// TIA Portal project "TIA_PORTAL_SORTING_STATION" (V20)

(* hardware
DEVICE "S7-1200 station_1"  S7-1200 Station
   slot 0: "Rack_0"  S7-1200 Rack  Rack  V1.0
   slot 1: "PLC_1"  CPU 1214C AC/DC/Rly  6ES7 214-1BG40-0XB0  V4.1
*)

// ===== PLC "PLC_1"  CPU 1214C AC/DC/Rly =====

VAR_GLOBAL   // PLC tag table "Default tag table"
   "Sensor_Pieza" AT %I0.0 : Bool;
   "CINTA" AT %Q0.0 : Bool;
   "S_LASER_RAMPA" AT %I0.2 : Bool;
   "Llave" AT %I0.7 : Bool;
   "START" AT %I1.2 : Bool;
   "M_STARTING" AT %M2.1 : Bool;
   "SENSOR_SERVO1" AT %I0.1 : Bool;
   "SENSOR_SERVO2" AT %I0.3 : Bool;
   "System_Byte" AT %MB300 : Byte;
   "FirstScan" AT %M300.0 : Bool;
   "DiagStatusUpdate" AT %M300.1 : Bool;
   "AlwaysTRUE" AT %M300.2 : Bool;
   "AlwaysFALSE" AT %M300.3 : Bool;
   "SIEMPRE_CERO" AT %M0.0 : Bool;
   "SIEMPRE_UNO" AT %M0.1 : Bool;
   "M_STOPPED" AT %M2.0 : Bool;
   "M_STARTED" AT %M2.2 : Bool;
   "M_STOPPING" AT %M2.3 : Bool;
   "M_ABORTING" AT %M2.4 : Bool;
   "M_RESET" AT %M2.5 : Bool;
   "M_FIN_CICLO" AT %M2.6 : Bool;
   "RESET" AT %I1.1 : Bool;
   "STOP" AT %I1.0 : Bool;
   "IR_A_M_STOPPED" AT %M4.3 : Bool;
   "PILOTO_START" AT %Q0.4 : Bool;
   "PILOTO_RESET" AT %Q0.5 : Bool;
   "Q1_STOPPED" AT %Q0.6 : Bool;
   "Q2_EMEG" AT %Q0.7 : Bool;
   "Timer_1" AT %M5.0 : Bool;
   "Tag_3" AT %M6.0 : Bool;
   "Intermitente" AT %M6.1 : Bool;
   "M_CINTA" AT %M3.0 : Bool;
   "Tag_1" AT %MB3 : Byte;
   "M_INICIO_RESET" AT %M4.2 : Bool;
   "M_FIN_RESET" AT %M4.1 : Bool;
   "M_SERVO_1" AT %M3.1 : Bool;
   "M_SERVO_2" AT %M3.2 : Bool;
   "M_PISTON" AT %M3.3 : Bool;
   "START_TIMER" AT %M5.1 : Bool;
   "M_INICIO_SECUENCIA" AT %M3.4 : Bool;
   "S_BARRERA" AT %I0.6 : Bool;
   "S_CANCELA_NEGRO" AT %I0.5 : Bool;
   "S_PIEZA_METALICA" AT %I0.4 : Bool;
   "SERVO_1" AT %Q0.1 : Bool;
   "SERVO_2" AT %Q0.2 : Bool;
   "PISTON" AT %Q0.3 : Bool;
   "M_PIEZA" AT %M3.5 : Bool;
   "Tag_2" AT %MW100 : Int;
   "M_TOTAL_ROJO" AT %M2.7 : Bool;
   "M_TOTAL_METAL" AT %M4.0 : Bool;
   "Tag_4" AT %MW101 : Int;
   "M_ROJO" AT %M7.0 : Bool;
   "M_BANDA_R" AT %M7.1 : Bool;
   "Tag_5" AT %MW102 : Int;
   "Tag_6" AT %MW107 : Int;
   "Tag_7" AT %MB7 : Byte;
   "Tag_8" AT %MB4 : Byte;
   "Tag_9" AT %MB5 : Byte;
   "M_Negro" AT %M7.2 : Bool;
END_VAR

VAR_GLOBAL   // PLC tag table "Tag table_1"
   "Clock_Byte" AT %MB100 : Byte;
   "Clock_10Hz" AT %M100.0 : Bool;
   "Clock_5Hz" AT %M100.1 : Bool;
   "Clock_2.5Hz" AT %M100.2 : Bool;
   "Clock_2Hz" AT %M100.3 : Bool;
   "Clock_1.25Hz" AT %M100.4 : Bool;
   "Clock_1Hz" AT %M100.5 : Bool;
   "Clock_0.625Hz" AT %M100.6 : Bool;
   "Clock_0.5Hz" AT %M100.7 : Bool;
END_VAR

// folder: System blocks/Program resources

DATA_BLOCK "IEC_Timer_0_DB"   // DB1
{ S7_Optimized_Access := 'TRUE' }
AUTHOR : Simatic
FAMILY : IEC
NAME : IEC_TMR
VERSION : 1.0
// stored: InstanceOfName IEC_TIMER
"IEC_TIMER"
BEGIN
END_DATA_BLOCK

DATA_BLOCK "IEC_Timer_0_DB_1"   // DB2
{ S7_Optimized_Access := 'TRUE' }
AUTHOR : Simatic
FAMILY : IEC
NAME : IEC_TMR
VERSION : 1.0
// stored: InstanceOfName IEC_TIMER
"IEC_TIMER"
BEGIN
END_DATA_BLOCK

DATA_BLOCK "IEC_Timer_0_DB_2"   // DB3
{ S7_Optimized_Access := 'TRUE' }
AUTHOR : Simatic
FAMILY : IEC
NAME : IEC_TMR
VERSION : 1.0
// stored: InstanceOfName IEC_TIMER
"IEC_TIMER"
BEGIN
END_DATA_BLOCK

DATA_BLOCK "IEC_Timer_0_DB_3"   // DB4
{ S7_Optimized_Access := 'TRUE' }
AUTHOR : Simatic
FAMILY : IEC
NAME : IEC_TMR
VERSION : 1.0
// stored: InstanceOfName IEC_TIMER
"IEC_TIMER"
BEGIN
END_DATA_BLOCK

DATA_BLOCK "IEC_Timer_0_DB_4"   // DB5
{ S7_Optimized_Access := 'TRUE' }
AUTHOR : Simatic
FAMILY : IEC
NAME : IEC_TMR
VERSION : 1.0
// stored: InstanceOfName IEC_TIMER
"IEC_TIMER"
BEGIN
END_DATA_BLOCK

DATA_BLOCK "IEC_Timer_0_DB_5"   // DB6
{ S7_Optimized_Access := 'TRUE' }
AUTHOR : Simatic
FAMILY : IEC
NAME : IEC_TMR
VERSION : 1.0
// stored: InstanceOfName IEC_TIMER
"IEC_TIMER"
BEGIN
END_DATA_BLOCK

DATA_BLOCK "IEC_Timer_0_DB_6"   // DB7
{ S7_Optimized_Access := 'TRUE' }
AUTHOR : Simatic
FAMILY : IEC
NAME : IEC_TMR
VERSION : 1.0
// stored: InstanceOfName IEC_TIMER
"IEC_TIMER"
BEGIN
END_DATA_BLOCK

DATA_BLOCK "IEC_Timer_0_DB_7"   // DB8
{ S7_Optimized_Access := 'TRUE' }
AUTHOR : Simatic
FAMILY : IEC
NAME : IEC_TMR
VERSION : 1.0
// stored: InstanceOfName IEC_TIMER
"IEC_TIMER"
BEGIN
END_DATA_BLOCK

DATA_BLOCK "IEC_Counter_0_DB"   // DB10
{ S7_Optimized_Access := 'TRUE' }
AUTHOR : Simatic
FAMILY : IEC
NAME : CNTR
VERSION : 1.0
// stored: InstanceOfName IEC_COUNTER
"IEC_COUNTER"
BEGIN
END_DATA_BLOCK

DATA_BLOCK "IEC_Counter_0_DB_1"   // DB11
{ S7_Optimized_Access := 'TRUE' }
AUTHOR : Simatic
FAMILY : IEC
NAME : CNTR
VERSION : 1.0
// stored: InstanceOfName IEC_COUNTER
"IEC_COUNTER"
BEGIN
END_DATA_BLOCK

DATA_BLOCK "IEC_Counter_0_DB_2"   // DB12
{ S7_Optimized_Access := 'TRUE' }
AUTHOR : Simatic
FAMILY : IEC
NAME : CNTR
VERSION : 1.0
// stored: InstanceOfName IEC_COUNTER
"IEC_COUNTER"
BEGIN
END_DATA_BLOCK

// folder: (top level)

FUNCTION "RESET_ESTADO" : Void   // FC1, LAD
{ S7_Optimized_Access := 'TRUE' }
VERSION : 0.1
BEGIN

REGION Network 1
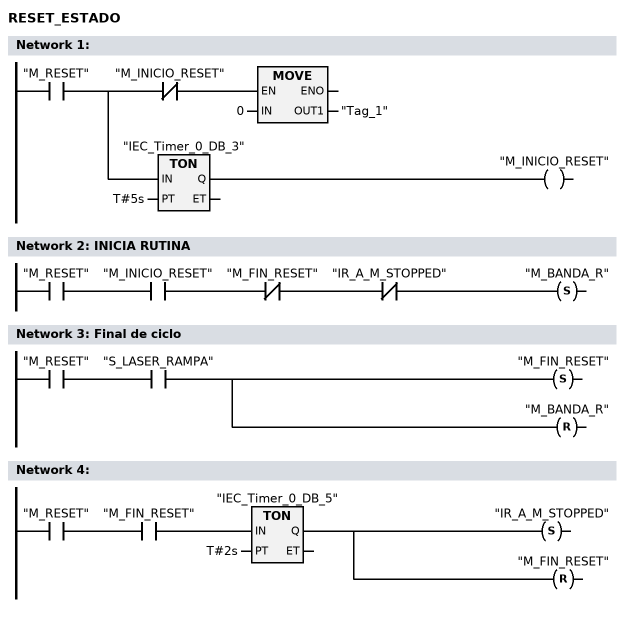
   IF "M_RESET" AND NOT "M_INICIO_RESET" THEN "Tag_1" := 0; END_IF;
   "IEC_Timer_0_DB_3".TON(IN := "M_RESET", PT := T#5s);
   "M_INICIO_RESET" := "IEC_Timer_0_DB_3".Q;
END_REGION

REGION Network 2: INICIA RUTINA
   RUNG wire#powerrail
      Contact( "M_RESET" )
      Contact( "M_INICIO_RESET" )
      I_Contact( "M_FIN_RESET" )
      I_Contact( "IR_A_M_STOPPED" )
      S_Coil( "M_BANDA_R" )
   END_RUNG
   // the same network as SCL:
   IF "M_RESET" AND "M_INICIO_RESET" AND NOT "M_FIN_RESET" AND NOT "IR_A_M_STOPPED" THEN
       "M_BANDA_R" := TRUE;
   END_IF;
END_REGION

REGION Network 3: Final de ciclo
   RUNG wire#powerrail
      Contact( "M_RESET" )
      Contact( "S_LASER_RAMPA" )
      wire#w1
      S_Coil( "M_FIN_RESET" )
   END_RUNG
   RUNG wire#w1
      R_Coil( "M_BANDA_R" )
   END_RUNG
   // the same network as SCL:
   IF "M_RESET" AND "S_LASER_RAMPA" THEN
       "M_FIN_RESET" := TRUE;
       "M_BANDA_R" := FALSE;
   END_IF;
END_REGION

REGION Network 4
   "IEC_Timer_0_DB_5".TON(IN := "M_RESET" AND "M_FIN_RESET", PT := T#2s);
   IF "IEC_Timer_0_DB_5".Q THEN
       "IR_A_M_STOPPED" := TRUE;
       "M_FIN_RESET" := FALSE;
   END_IF;
END_REGION
END_FUNCTION

FUNCTION "Maquina_Estado" : Void   // FC2, LAD
{ S7_Optimized_Access := 'TRUE' }
VERSION : 0.1
   VAR_TEMP   // added for the SCL form of the ladder/FBD networks
      _w1 : Bool;
   END_VAR
BEGIN

REGION Network 1: SECUENCIA_STARTING
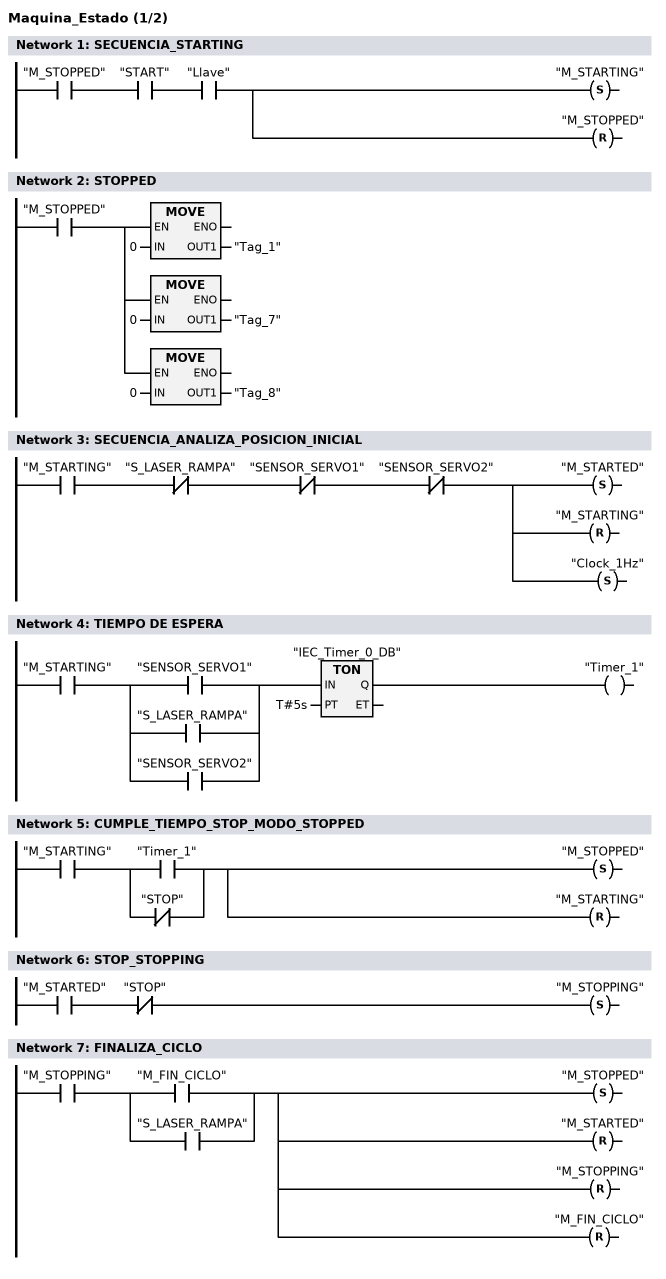
   RUNG wire#powerrail
      Contact( "M_STOPPED" )
      Contact( "START" )
      Contact( "Llave" )
      wire#w1
      S_Coil( "M_STARTING" )
   END_RUNG
   RUNG wire#w1
      R_Coil( "M_STOPPED" )
   END_RUNG
   // the same network as SCL:
   IF "M_STOPPED" AND "START" AND "Llave" THEN
       "M_STARTING" := TRUE;
       "M_STOPPED" := FALSE;
   END_IF;
END_REGION

REGION Network 2: STOPPED
   RUNG wire#powerrail
      Contact( "M_STOPPED" )
      wire#w1
      Move(in := 0, out1 => "Tag_1")
   END_RUNG
   RUNG wire#w1
      Move(in := 0, out1 => "Tag_7")
   END_RUNG
   RUNG wire#w1
      Move(in := 0, out1 => "Tag_8")
   END_RUNG
   // the same network as SCL:
   IF "M_STOPPED" THEN
       "Tag_1" := 0;
       "Tag_7" := 0;
       "Tag_8" := 0;
   END_IF;
END_REGION

REGION Network 3: SECUENCIA_ANALIZA_POSICION_INICIAL
   RUNG wire#powerrail
      Contact( "M_STARTING" )
      I_Contact( "S_LASER_RAMPA" )
      I_Contact( "SENSOR_SERVO1" )
      I_Contact( "SENSOR_SERVO2" )
      wire#w1
      S_Coil( "M_STARTED" )
   END_RUNG
   RUNG wire#w1
      R_Coil( "M_STARTING" )
   END_RUNG
   RUNG wire#w1
      S_Coil( "Clock_1Hz" )
   END_RUNG
   // the same network as SCL:
   IF "M_STARTING" AND NOT "S_LASER_RAMPA" AND NOT "SENSOR_SERVO1" AND NOT "SENSOR_SERVO2" THEN
       "M_STARTED" := TRUE;
   END_IF;
   #_w1 := "M_STARTING" AND NOT "S_LASER_RAMPA" AND NOT "SENSOR_SERVO1" AND NOT "SENSOR_SERVO2";
   IF #_w1 THEN
       "M_STARTING" := FALSE;
       "Clock_1Hz" := TRUE;
   END_IF;
END_REGION

REGION Network 4: TIEMPO DE ESPERA
   "IEC_Timer_0_DB".TON(IN := "M_STARTING" AND ("SENSOR_SERVO1" OR "S_LASER_RAMPA" OR "SENSOR_SERVO2"),
                        PT := T#5s);
   "Timer_1" := "IEC_Timer_0_DB".Q;
END_REGION

REGION Network 5: CUMPLE_TIEMPO_STOP_MODO_STOPPED
   RUNG wire#powerrail
      Contact( "M_STARTING" )
      wire#w1
      Contact( "Timer_1" )
      wire#w2
      S_Coil( "M_STOPPED" )
   END_RUNG
   RUNG wire#w1
      I_Contact( "STOP" )
   END_RUNG wire#w2
   RUNG wire#w2
      R_Coil( "M_STARTING" )
   END_RUNG
   // the same network as SCL:
   IF "M_STARTING" AND ("Timer_1" OR NOT "STOP") THEN
       "M_STOPPED" := TRUE;
       "M_STARTING" := FALSE;
   END_IF;
END_REGION

REGION Network 6: STOP_STOPPING
   RUNG wire#powerrail
      Contact( "M_STARTED" )
      I_Contact( "STOP" )
      S_Coil( "M_STOPPING" )
   END_RUNG
   // the same network as SCL:
   IF "M_STARTED" AND NOT "STOP" THEN "M_STOPPING" := TRUE; END_IF;
END_REGION

REGION Network 7: FINALIZA_CICLO
   RUNG wire#powerrail
      Contact( "M_STOPPING" )
      wire#w1
      Contact( "M_FIN_CICLO" )
      wire#w2
      S_Coil( "M_STOPPED" )
   END_RUNG
   RUNG wire#w1
      Contact( "S_LASER_RAMPA" )
   END_RUNG wire#w2
   RUNG wire#w2
      R_Coil( "M_STARTED" )
   END_RUNG
   RUNG wire#w2
      R_Coil( "M_STOPPING" )
   END_RUNG
   RUNG wire#w2
      R_Coil( "M_FIN_CICLO" )
   END_RUNG
   // the same network as SCL:
   IF "M_STOPPING" AND ("M_FIN_CICLO" OR "S_LASER_RAMPA") THEN
       "M_STOPPED" := TRUE;
       "M_STARTED" := FALSE;
   END_IF;
   #_w1 := "M_STOPPING" AND ("M_FIN_CICLO" OR "S_LASER_RAMPA");
   IF #_w1 THEN
       "M_STOPPING" := FALSE;
       "M_FIN_CICLO" := FALSE;
   END_IF;
END_REGION

REGION Network 8: SI PRESIONA EL PARO DE EMERGENCIA PASAMOS A ABORTING
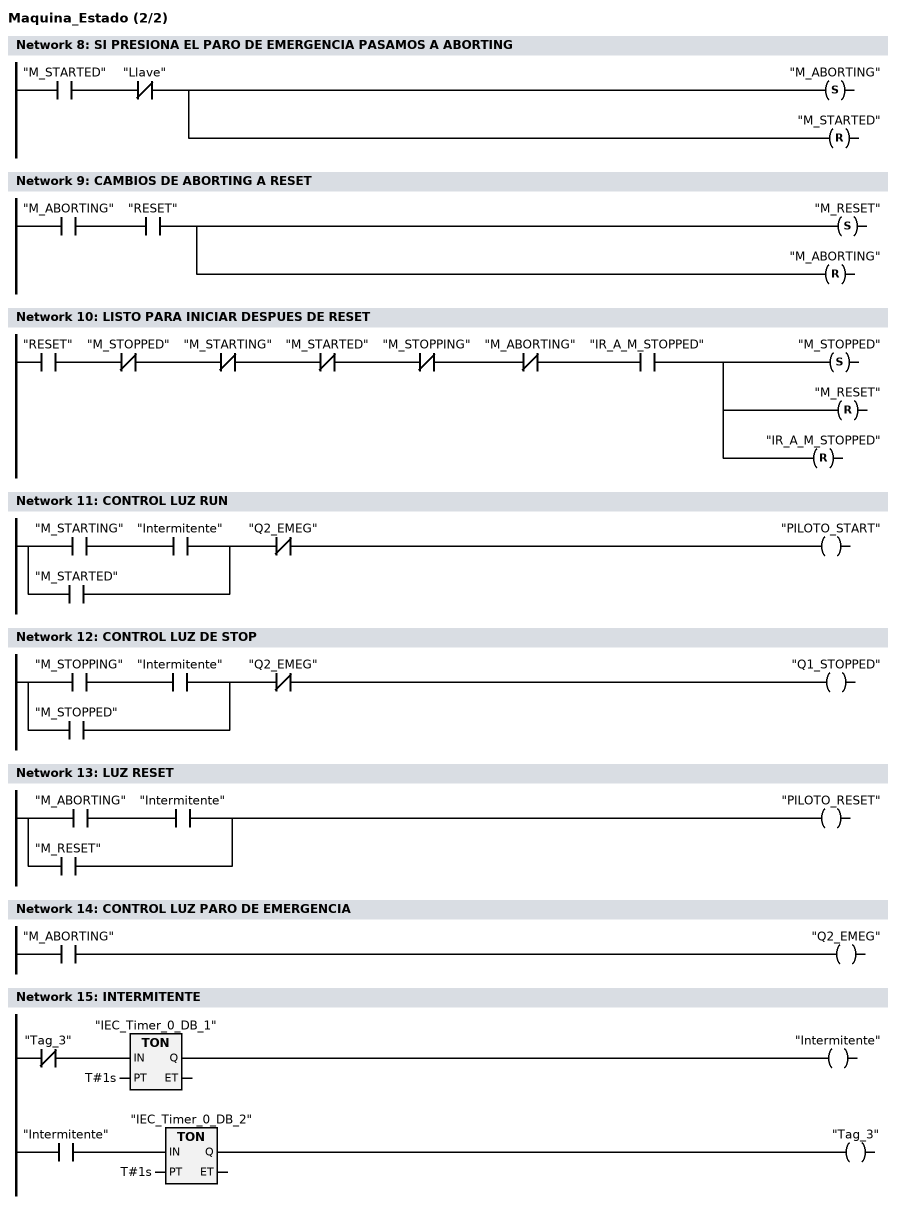
   RUNG wire#powerrail
      Contact( "M_STARTED" )
      I_Contact( "Llave" )
      wire#w1
      S_Coil( "M_ABORTING" )
   END_RUNG
   RUNG wire#w1
      R_Coil( "M_STARTED" )
   END_RUNG
   // the same network as SCL:
   IF "M_STARTED" AND NOT "Llave" THEN
       "M_ABORTING" := TRUE;
       "M_STARTED" := FALSE;
   END_IF;
END_REGION

REGION Network 9: CAMBIOS DE ABORTING A RESET
   RUNG wire#powerrail
      Contact( "M_ABORTING" )
      Contact( "RESET" )
      wire#w1
      S_Coil( "M_RESET" )
   END_RUNG
   RUNG wire#w1
      R_Coil( "M_ABORTING" )
   END_RUNG
   // the same network as SCL:
   IF "M_ABORTING" AND "RESET" THEN
       "M_RESET" := TRUE;
       "M_ABORTING" := FALSE;
   END_IF;
END_REGION

REGION Network 10: LISTO PARA INICIAR DESPUES DE RESET
   RUNG wire#powerrail
      Contact( "RESET" )
      I_Contact( "M_STOPPED" )
      I_Contact( "M_STARTING" )
      I_Contact( "M_STARTED" )
      I_Contact( "M_STOPPING" )
      I_Contact( "M_ABORTING" )
      Contact( "IR_A_M_STOPPED" )
      wire#w1
      S_Coil( "M_STOPPED" )
   END_RUNG
   RUNG wire#w1
      R_Coil( "M_RESET" )
   END_RUNG
   RUNG wire#w1
      R_Coil( "IR_A_M_STOPPED" )
   END_RUNG
   // the same network as SCL:
   #_w1 := "RESET" AND NOT "M_STOPPED" AND NOT "M_STARTING" AND NOT "M_STARTED" AND NOT "M_STOPPING" AND NOT "M_ABORTING" AND "IR_A_M_STOPPED";
   IF #_w1 THEN
       "M_STOPPED" := TRUE;
       "M_RESET" := FALSE;
       "IR_A_M_STOPPED" := FALSE;
   END_IF;
END_REGION

REGION Network 11: CONTROL LUZ RUN
   RUNG wire#powerrail
      Contact( "M_STARTING" )
      Contact( "Intermitente" )
      wire#w1
      I_Contact( "Q2_EMEG" )
      Coil( "PILOTO_START" )
   END_RUNG
   RUNG wire#powerrail
      Contact( "M_STARTED" )
   END_RUNG wire#w1
   // the same network as SCL:
   "PILOTO_START" := (("M_STARTING" AND "Intermitente") OR "M_STARTED") AND NOT "Q2_EMEG";
END_REGION

REGION Network 12: CONTROL LUZ DE STOP
   RUNG wire#powerrail
      Contact( "M_STOPPING" )
      Contact( "Intermitente" )
      wire#w1
      I_Contact( "Q2_EMEG" )
      Coil( "Q1_STOPPED" )
   END_RUNG
   RUNG wire#powerrail
      Contact( "M_STOPPED" )
   END_RUNG wire#w1
   // the same network as SCL:
   "Q1_STOPPED" := (("M_STOPPING" AND "Intermitente") OR "M_STOPPED") AND NOT "Q2_EMEG";
END_REGION

REGION Network 13: LUZ RESET
   RUNG wire#powerrail
      Contact( "M_ABORTING" )
      Contact( "Intermitente" )
      wire#w1
      Coil( "PILOTO_RESET" )
   END_RUNG
   RUNG wire#powerrail
      Contact( "M_RESET" )
   END_RUNG wire#w1
   // the same network as SCL:
   "PILOTO_RESET" := ("M_ABORTING" AND "Intermitente") OR "M_RESET";
END_REGION

REGION Network 14: CONTROL LUZ PARO DE EMERGENCIA
   RUNG wire#powerrail
      Contact( "M_ABORTING" )
      Coil( "Q2_EMEG" )
   END_RUNG
   // the same network as SCL:
   "Q2_EMEG" := "M_ABORTING";
END_REGION

REGION Network 15: INTERMITENTE
   "IEC_Timer_0_DB_1".TON(IN := NOT "Tag_3", PT := T#1s);
   "Intermitente" := "IEC_Timer_0_DB_1".Q;
   "IEC_Timer_0_DB_2".TON(IN := "Intermitente", PT := T#1s);
   "Tag_3" := "IEC_Timer_0_DB_2".Q;
END_REGION
END_FUNCTION

FUNCTION "Programacion secuencia" : Void   // FC3, LAD
{ S7_Optimized_Access := 'TRUE' }
VERSION : 0.1
   VAR_TEMP   // added for the SCL form of the ladder/FBD networks
      _w1 : Bool;
   END_VAR
BEGIN

REGION Network 1: Comprobacion
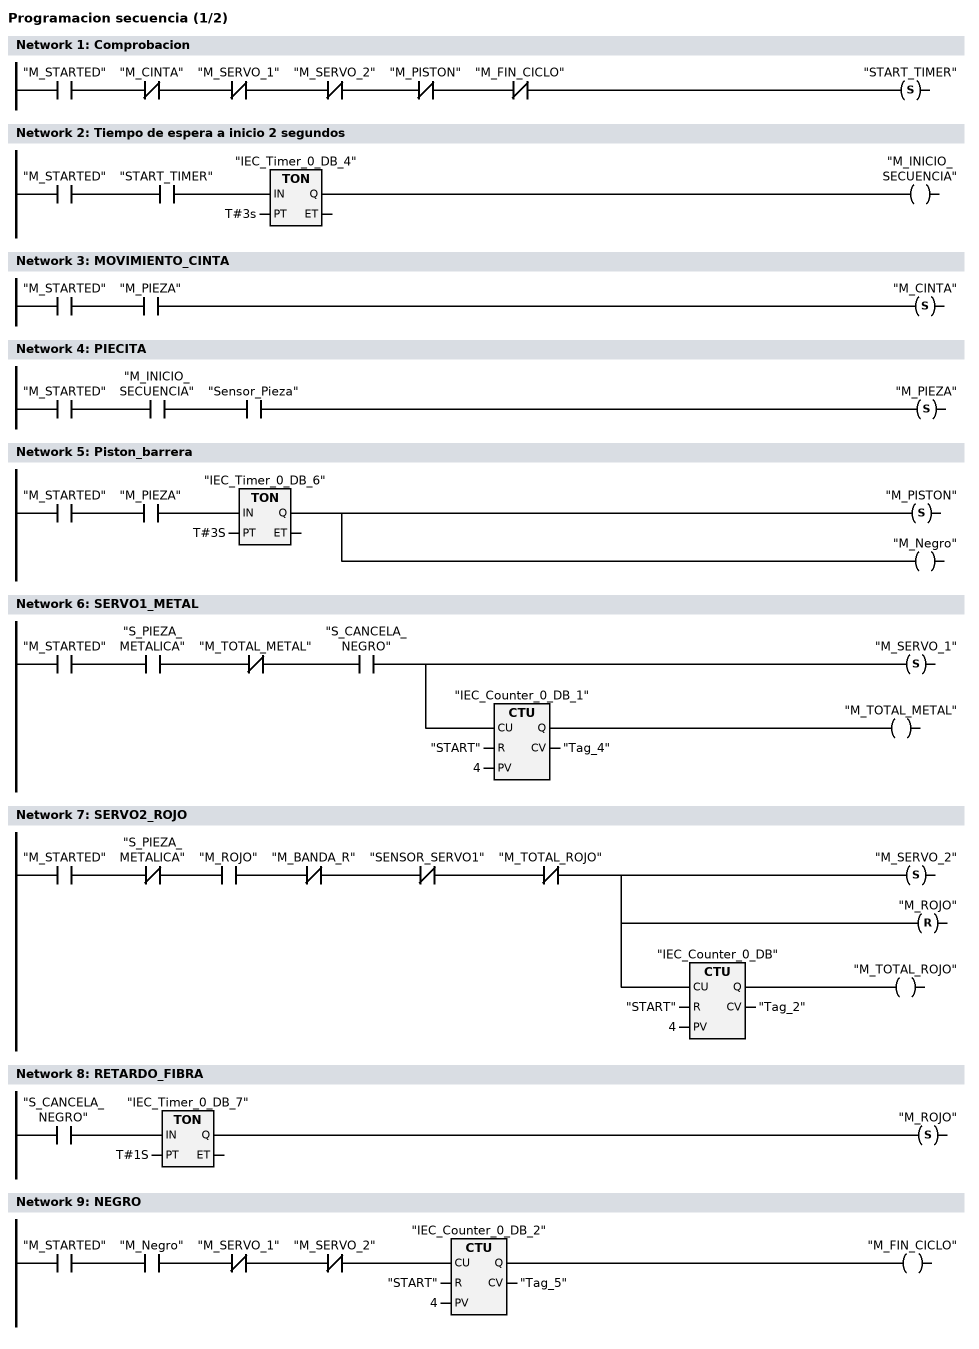
   RUNG wire#powerrail
      Contact( "M_STARTED" )
      I_Contact( "M_CINTA" )
      I_Contact( "M_SERVO_1" )
      I_Contact( "M_SERVO_2" )
      I_Contact( "M_PISTON" )
      I_Contact( "M_FIN_CICLO" )
      S_Coil( "START_TIMER" )
   END_RUNG
   // the same network as SCL:
   IF "M_STARTED" AND NOT "M_CINTA" AND NOT "M_SERVO_1" AND NOT "M_SERVO_2" AND NOT "M_PISTON" AND NOT "M_FIN_CICLO" THEN
       "START_TIMER" := TRUE;
   END_IF;
END_REGION

REGION Network 2: Tiempo de espera a inicio 2 segundos
   "IEC_Timer_0_DB_4".TON(IN := "M_STARTED" AND "START_TIMER", PT := T#3s);
   "M_INICIO_SECUENCIA" := "IEC_Timer_0_DB_4".Q;
END_REGION

REGION Network 3: MOVIMIENTO_CINTA
   RUNG wire#powerrail
      Contact( "M_STARTED" )
      Contact( "M_PIEZA" )
      S_Coil( "M_CINTA" )
   END_RUNG
   // the same network as SCL:
   IF "M_STARTED" AND "M_PIEZA" THEN "M_CINTA" := TRUE; END_IF;
END_REGION

REGION Network 4: PIECITA
   RUNG wire#powerrail
      Contact( "M_STARTED" )
      Contact( "M_INICIO_SECUENCIA" )
      Contact( "Sensor_Pieza" )
      S_Coil( "M_PIEZA" )
   END_RUNG
   // the same network as SCL:
   IF "M_STARTED" AND "M_INICIO_SECUENCIA" AND "Sensor_Pieza" THEN "M_PIEZA" := TRUE; END_IF;
END_REGION

REGION Network 5: Piston_barrera
   "IEC_Timer_0_DB_6".TON(IN := "M_STARTED" AND "M_PIEZA", PT := T#3S);
   IF "IEC_Timer_0_DB_6".Q THEN "M_PISTON" := TRUE; END_IF;
   "M_Negro" := "IEC_Timer_0_DB_6".Q;
END_REGION

REGION Network 6: SERVO1_METAL
   #_w1 := "M_STARTED" AND "S_PIEZA_METALICA" AND NOT "M_TOTAL_METAL" AND "S_CANCELA_NEGRO";
   IF #_w1 THEN "M_SERVO_1" := TRUE; END_IF;
   "IEC_Counter_0_DB_1".CTU(CU := #_w1, R := "START", PV := 4, CV => "Tag_4");
   "M_TOTAL_METAL" := "IEC_Counter_0_DB_1".Q;
END_REGION

REGION Network 7: SERVO2_ROJO
   #_w1 := "M_STARTED" AND NOT "S_PIEZA_METALICA" AND "M_ROJO" AND NOT "M_BANDA_R" AND NOT "SENSOR_SERVO1" AND NOT "M_TOTAL_ROJO";
   IF #_w1 THEN
       "M_SERVO_2" := TRUE;
       "M_ROJO" := FALSE;
   END_IF;
   "IEC_Counter_0_DB".CTU(CU := #_w1, R := "START", PV := 4, CV => "Tag_2");
   "M_TOTAL_ROJO" := "IEC_Counter_0_DB".Q;
END_REGION

REGION Network 8: RETARDO_FIBRA
   "IEC_Timer_0_DB_7".TON(IN := "S_CANCELA_NEGRO", PT := T#1S);
   IF "IEC_Timer_0_DB_7".Q THEN "M_ROJO" := TRUE; END_IF;
END_REGION

REGION Network 9: NEGRO
   "IEC_Counter_0_DB_2".CTU(CU := "M_STARTED" AND "M_Negro" AND NOT "M_SERVO_1" AND NOT "M_SERVO_2",
                           R := "START",
                           PV := 4,
                           CV => "Tag_5");
   "M_FIN_CICLO" := "IEC_Counter_0_DB_2".Q;
END_REGION

REGION Network 10: SI ESTA STOPING
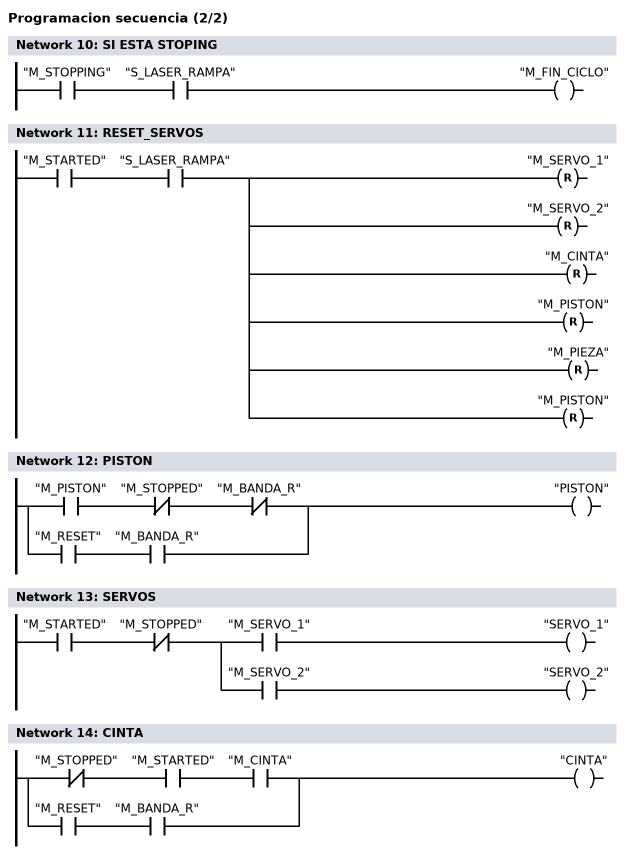
   RUNG wire#powerrail
      Contact( "M_STOPPING" )
      Contact( "S_LASER_RAMPA" )
      Coil( "M_FIN_CICLO" )
   END_RUNG
   // the same network as SCL:
   "M_FIN_CICLO" := "M_STOPPING" AND "S_LASER_RAMPA";
END_REGION

REGION Network 11: RESET_SERVOS
   RUNG wire#powerrail
      Contact( "M_STARTED" )
      Contact( "S_LASER_RAMPA" )
      wire#w1
      R_Coil( "M_SERVO_1" )
   END_RUNG
   RUNG wire#w1
      R_Coil( "M_SERVO_2" )
   END_RUNG
   RUNG wire#w1
      R_Coil( "M_CINTA" )
   END_RUNG
   RUNG wire#w1
      R_Coil( "M_PISTON" )
   END_RUNG
   RUNG wire#w1
      R_Coil( "M_PIEZA" )
   END_RUNG
   RUNG wire#w1
      R_Coil( "M_PISTON" )
   END_RUNG
   // the same network as SCL:
   IF "M_STARTED" AND "S_LASER_RAMPA" THEN
       "M_SERVO_1" := FALSE;
       "M_SERVO_2" := FALSE;
       "M_CINTA" := FALSE;
       "M_PISTON" := FALSE;
       "M_PIEZA" := FALSE;
       "M_PISTON" := FALSE;
   END_IF;
END_REGION

REGION Network 12: PISTON
   RUNG wire#powerrail
      Contact( "M_PISTON" )
      I_Contact( "M_STOPPED" )
      I_Contact( "M_BANDA_R" )
      wire#w1
      Coil( "PISTON" )
   END_RUNG
   RUNG wire#powerrail
      Contact( "M_RESET" )
      Contact( "M_BANDA_R" )
   END_RUNG wire#w1
   // the same network as SCL:
   "PISTON" := ("M_PISTON" AND NOT "M_STOPPED" AND NOT "M_BANDA_R") OR ("M_RESET" AND "M_BANDA_R");
END_REGION

REGION Network 13: SERVOS
   RUNG wire#powerrail
      Contact( "M_STARTED" )
      I_Contact( "M_STOPPED" )
      wire#w1
      Contact( "M_SERVO_1" )
      Coil( "SERVO_1" )
   END_RUNG
   RUNG wire#w1
      Contact( "M_SERVO_2" )
      Coil( "SERVO_2" )
   END_RUNG
   // the same network as SCL:
   #_w1 := "M_STARTED" AND NOT "M_STOPPED";
   "SERVO_1" := #_w1 AND "M_SERVO_1";
   "SERVO_2" := #_w1 AND "M_SERVO_2";
END_REGION

REGION Network 14: CINTA
   RUNG wire#powerrail
      I_Contact( "M_STOPPED" )
      Contact( "M_STARTED" )
      Contact( "M_CINTA" )
      wire#w1
      Coil( "CINTA" )
   END_RUNG
   RUNG wire#powerrail
      Contact( "M_RESET" )
      Contact( "M_BANDA_R" )
   END_RUNG wire#w1
   // the same network as SCL:
   "CINTA" := (NOT "M_STOPPED" AND "M_STARTED" AND "M_CINTA") OR ("M_RESET" AND "M_BANDA_R");
END_REGION
END_FUNCTION

ORGANIZATION_BLOCK "Main"   // OB1, LAD, ProgramCycle
TITLE = "Main Program Sweep (Cycle)"
{ S7_Optimized_Access := 'TRUE' }
VERSION : 0.1
   VAR_INPUT
      Initial_Call : Bool;   // Initial call of this OB
      Remanence : Bool;   // =True, if remanent data are available
   END_VAR
BEGIN

REGION Network 1: Maquina_Estado
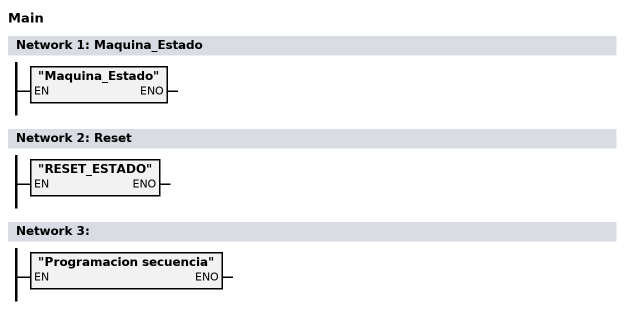
   RUNG wire#powerrail
      "Maquina_Estado"()
   END_RUNG
   // the same network as SCL:
   "Maquina_Estado"();
END_REGION

REGION Network 2: Reset
   RUNG wire#powerrail
      "RESET_ESTADO"()
   END_RUNG
   // the same network as SCL:
   "RESET_ESTADO"();
END_REGION

REGION Network 3
   RUNG wire#powerrail
      "Programacion secuencia"()
   END_RUNG
   // the same network as SCL:
   "Programacion secuencia"();
END_REGION
END_ORGANIZATION_BLOCK

ORGANIZATION_BLOCK "Startup"   // OB100, LAD, Startup
TITLE = "Complete Restart"
{ S7_Optimized_Access := 'TRUE' }
VERSION : 0.1
   VAR_INPUT
      LostRetentive : Bool;   // True if retentive data are lost
      LostRTC : Bool;   // True if date and time are lost
   END_VAR
BEGIN

REGION Network 1
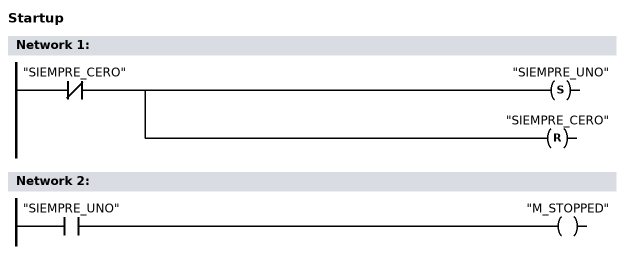
   RUNG wire#powerrail
      I_Contact( "SIEMPRE_CERO" )
      wire#w1
      S_Coil( "SIEMPRE_UNO" )
   END_RUNG
   RUNG wire#w1
      R_Coil( "SIEMPRE_CERO" )
   END_RUNG
   // the same network as SCL:
   IF NOT "SIEMPRE_CERO" THEN
       "SIEMPRE_UNO" := TRUE;
       "SIEMPRE_CERO" := FALSE;
   END_IF;
END_REGION

REGION Network 2
   RUNG wire#powerrail
      Contact( "SIEMPRE_UNO" )
      Coil( "M_STOPPED" )
   END_RUNG
   // the same network as SCL:
   "M_STOPPED" := "SIEMPRE_UNO";
END_REGION
END_ORGANIZATION_BLOCK